(* IEC 61131-3 sources: plc_generation_empirical_study/datasets/task_bank_c04_reverse_runtime_v0_3/tasks/C04_S12_lean_composite/negative_control, 1 file *)

(* ---- NC1.st ---- *)
FUNCTION_BLOCK C04_S12_lean_composite
VAR_INPUT
    A_S1 : BOOL;
    A_S2 : BOOL;
    A_S3 : BOOL;
    B_EventA : BOOL;
    B_EventB : BOOL;
    B_Arm : BOOL;
    B_Reset : BOOL;
    SubsystemBEnable : BOOL;
    CrossReset : BOOL;
END_VAR
VAR_OUTPUT
    A_Vote : BOOL;
    A_Unanimous : BOOL;
    B_Captured : BOOL;
    B_Code : INT;
    B_Pulse : BOOL;
    CrossReady : BOOL;
    CrossBlocked : BOOL;
END_VAR
VAR
    B_PrevA : BOOL := FALSE;
    B_PrevB : BOOL := FALSE;
END_VAR

A_Vote := (A_S1 AND A_S2) OR (A_S1 AND A_S3) OR (A_S2 AND A_S3);
A_Unanimous := (A_S1 AND A_S2 AND A_S3) OR ((NOT A_S1) AND (NOT A_S2) AND (NOT A_S3));

IF CrossReset THEN
    CrossReady := FALSE;
ELSIF A_Vote THEN
    CrossReady := TRUE;
END_IF;
CrossBlocked := FALSE;

IF SubsystemBEnable AND CrossReady THEN
    B_Pulse := FALSE;
    IF B_Reset THEN
        B_Captured := FALSE;
        B_Code := 0;
    ELSIF B_Arm AND (NOT B_Captured) THEN
        IF B_EventA AND (NOT B_PrevA) THEN
            B_Captured := TRUE;
            B_Code := 1;
            B_Pulse := TRUE;
        ELSIF B_EventB AND (NOT B_PrevB) THEN
            B_Captured := TRUE;
            B_Code := 2;
            B_Pulse := TRUE;
        END_IF;
    END_IF;
    B_PrevA := B_EventA;
    B_PrevB := B_EventB;
ELSE
    B_Captured := FALSE;
    B_Code := 0;
    B_Pulse := FALSE;
END_IF;

END_FUNCTION_BLOCK
